PROGRAM MAIN
VAR
	
END_VAR

P_Example_1();
P_Example_2();

END_PROGRAM

(* stored: Version 1.1.0.1, ProductVersion 3.1.4024.4
   POU MAIN: Id {a8718cfc-9873-4f98-af26-d643b2d89a91}, SpecialFunc None *)
